TYPE ST_ConfiguredAlarmState :
STRUCT
	PreviousCondition : BOOL;
	Latched : BOOL;
	Active : BOOL;
	Acknowledged : BOOL;
	OccurrenceCount : UDINT;
	FirstOccurrenceDateTime : STRING(20);
END_STRUCT
END_TYPE

(* stored: Version 1.1.0.1, ProductVersion 3.1.4026.18
   DUT ST_ConfiguredAlarmState: Id {711ede85-7607-43f2-a233-271f83f2a8dc} *)
